(* PLC project Unnamed, Unknown Unnamed 1 *)
(* stored: creationDateTime 2021-04-23T13:43:33, modificationDateTime 2021-04-23T13:44:47 *)

PROGRAM VariablesConnections
  VAR
    InputVariable : DINT;
    Input/OutputVariable : DINT;
    OutputVariable : DINT;
  END_VAR

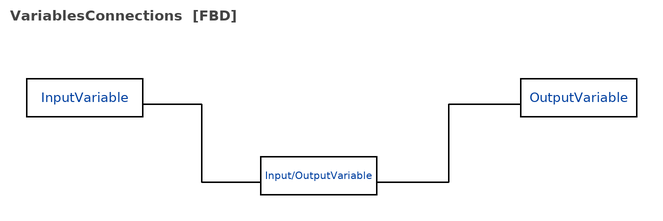
(* FBD diagram, written out as Structured Text *)
OutputVariable := Input/OutputVariable;
Input/OutputVariable := InputVariable;
END_PROGRAM

CONFIGURATION Config0
  RESOURCE Res0 ON PLC
    TASK task0(INTERVAL := T#20ms, PRIORITY := 0);
    PROGRAM instance0 WITH task0 : VariablesConnections;
  END_RESOURCE
END_CONFIGURATION
